Omron CX-Programmer project 新專案 (CX-Programmer 9.54)

# PLC 新PLC1: CJ2M CPU31
I/O table (CPU CJ2M-CPU31): rack 0 slot 0 CJ1W-SCU41-V1; rack 0 slot 1 CJ1W-ID231; rack 0 slot 2 CJ1W-ID231; rack 0 slot 3 CJ1W-OD231; rack 0 slot 4 CJ1W-ID211; rack 0 slot 11 CJ2M-EIP21

## Global symbols (name address type ; comment)
3.10 BOOL  ; SG舵機上感測器
3.11 BOOL  ; SG舵機下感測器
3.12 BOOL  ; PH舵機上感測器
3.13 BOOL  ; PH舵機下感測器
3.14 BOOL  ; UV舵機上感測器
3.15 BOOL  ; UV舵機下感測器
4.00 BOOL  ; SG隔膜清洗
4.01 BOOL  ; PH隔膜清洗
4.02 BOOL  ; UV隔膜清洗
4.03 BOOL  ; UV補純水
4.04 BOOL  ; SG抽液馬達
4.08 BOOL  ; 純水馬達
4.09 BOOL  ; SG舵機
4.10 BOOL  ; PH舵機
4.11 BOOL  ; UV舵機
4.12 BOOL  ; UV攪拌器
50.00 BOOL  ; 重置
50.01 BOOL  ; UV整數加
50.02 BOOL  ; UV分數加
50.03 BOOL  ; 六千
50.04 BOOL  ; 指定
50.05 BOOL  ; 回推
50.06 BOOL  ; 零點
50.07 BOOL  ; 方向
50.08 BOOL  ; 左轉
50.09 BOOL  ; 中間
50.10 BOOL  ; 右轉
50.11 BOOL  ; 速度
5.00 BOOL  ; 綠燈
5.01 BOOL  ; 橘燈
5.02 BOOL  ; 紅燈
5.03 BOOL  ; 蜂鳴器
6.00 BOOL  ; 純水低液位
6.01 BOOL  ; 純水高液位
D0 CHANNEL  ; Robot起點
D1 CHANNEL  ; Robot終點
D100 CHANNEL  ; SG平台狀態
D2 CHANNEL  ; Robot目前位置
D200 CHANNEL  ; PH平台狀態
D20001 CHANNEL  ; Seat1
D20002 CHANNEL  ; Seat2
D20003 CHANNEL  ; Seat3
D3 CHANNEL  ; 開蓋旗標
D300 CHANNEL  ; UV平台狀態
D301 CHANNEL  ; 針閥排隊
D310 CHANNEL  ; 針一狀態
D311 CHANNEL  ; 針一是否校正液
D312 CHANNEL  ; 針一整數次數
D313 CHANNEL  ; 針一分數高位
D314 CHANNEL  ; 針一分數低位
D315 CHANNEL  ; 針一指令傳送成功
D320 CHANNEL  ; 針二狀態
D321 CHANNEL  ; 針二是否校正液
D322 CHANNEL  ; 針二整數次數
D323 CHANNEL  ; 針二分數高位
D324 CHANNEL  ; 針二分數低位
D325 CHANNEL  ; 針二指令傳送成功
D330 CHANNEL  ; 針三狀態
D331 CHANNEL  ; 針三是否校正液
D332 CHANNEL  ; 針三整數次數
D333 CHANNEL  ; 針三分數高位
D334 CHANNEL  ; 針三分數低位
D335 CHANNEL  ; 針三指令傳送成功
D9998 CHANNEL  ; 稼動綠燈號
D9999 CHANNEL  ; 稼動率蜂鳴器
H100.00 BOOL  ; SG空閒
H100.01 BOOL  ; SG杯子送入
H100.02 BOOL  ; SG下舵機
H100.03 BOOL  ; SG抽樣品
H100.04 BOOL  ; SG等待
H100.05 BOOL  ; SG讀值中
H100.06 BOOL  ; SG起舵機
H100.07 BOOL  ; SG等移出
H100.08 BOOL  ; SG已移出
H100.09 BOOL  ; SG清洗
H100.10 BOOL  ; 清洗完畢
H150.01 BOOL  ; SG瓶子放入
H150.02 BOOL  ; SG下舵機
H150.03 BOOL  ; SG抽酸洗液
H150.04 BOOL  ; SG起舵機
H150.05 BOOL  ; SG等移出
H150.06 BOOL  ; SG已移出
H150.07 BOOL  ; SG清洗
H150.08 BOOL  ; SG清洗完畢
H200.00 BOOL  ; PH空閒
H200.01 BOOL  ; PH杯子送入
H200.02 BOOL  ; PH下舵機
H200.03 BOOL  ; PH等待
H200.04 BOOL  ; PH讀值中
H200.05 BOOL  ; PH起舵機
H200.06 BOOL  ; PH等移出
H200.07 BOOL  ; PH已移出
H200.08 BOOL  ; PH清洗
H200.09 BOOL  ; PH清洗完畢
H250.01 BOOL  ; PH水洗
H250.02 BOOL  ; PH水洗完畢
H300.00 BOOL  ; UV空閒
H300.01 BOOL  ; UV杯子送入
H300.02 BOOL  ; UV下舵機
H300.03 BOOL  ; UV樣品初始化
H300.04 BOOL  ; UV排液
H300.05 BOOL  ; UV注水
H300.06 BOOL  ; UV排乾
H300.07 BOOL  ; UV打歸零緩衝液
H300.08 BOOL  ; UV排液
H300.09 BOOL  ; UV等待
H300.10 BOOL  ; UV設定波長歸零
H300.11 BOOL  ; UV注水
H300.12 BOOL  ; UV排液
H300.13 BOOL  ; UV整數取樣
H300.14 BOOL  ; UV分數取樣
H300.15 BOOL  ; UV抽液
H301.00 BOOL  ; UV等待
H301.01 BOOL  ; UV讀值
H301.02 BOOL  ; UV起舵機
H301.03 BOOL  ; UV等待移出
H301.04 BOOL  ; UV已移出
H301.05 BOOL  ; UV針閥清洗
H301.06 BOOL  ; UV排乾
H301.07 BOOL  ; UV補水
H301.08 BOOL  ; UV排乾
H301.09 BOOL  ; UV清洗完畢
W0.00 BOOL  ; 針閥1初始化
W0.01 BOOL  ; 針閥二初始化
W300.00 BOOL  ; 樣品初始化開始
W300.01 BOOL  ; 樣品初始化中
W300.02 BOOL  ; 樣品初始化完成
W300.03 BOOL  ; 分數取樣完成
W301.00 BOOL  ; 打緩衝液開始
W301.01 BOOL  ; 打緩衝液中
W301.02 BOOL  ; 打緩衝液完成
W302.00 BOOL  ; UV整數取樣開始
W302.01 BOOL  ; UV整數取樣中
W302.02 BOOL  ; UV整數取樣完成
W303.00 BOOL  ; UV分數取樣開始
W303.01 BOOL  ; UV分數取樣中
W303.02 BOOL  ; UV分數取樣完成
W304.00 BOOL  ; 針閥清洗
W304.01 BOOL  ; 針閥清洗中
W304.02 BOOL  ; 針閥清洗完成
W304.03 BOOL  ; 補水
W305.00 BOOL  ; 二次補水
W305.01 BOOL  ; 三次補水
W306.00 BOOL  ; 清洗二次補水
W306.01 BOOL  ; 清洗三次補水

## Program 新增程式1 (cyclic task 0)
Local symbols
FFFF CHANNEL
md BOOL

### Section Platform1_SG

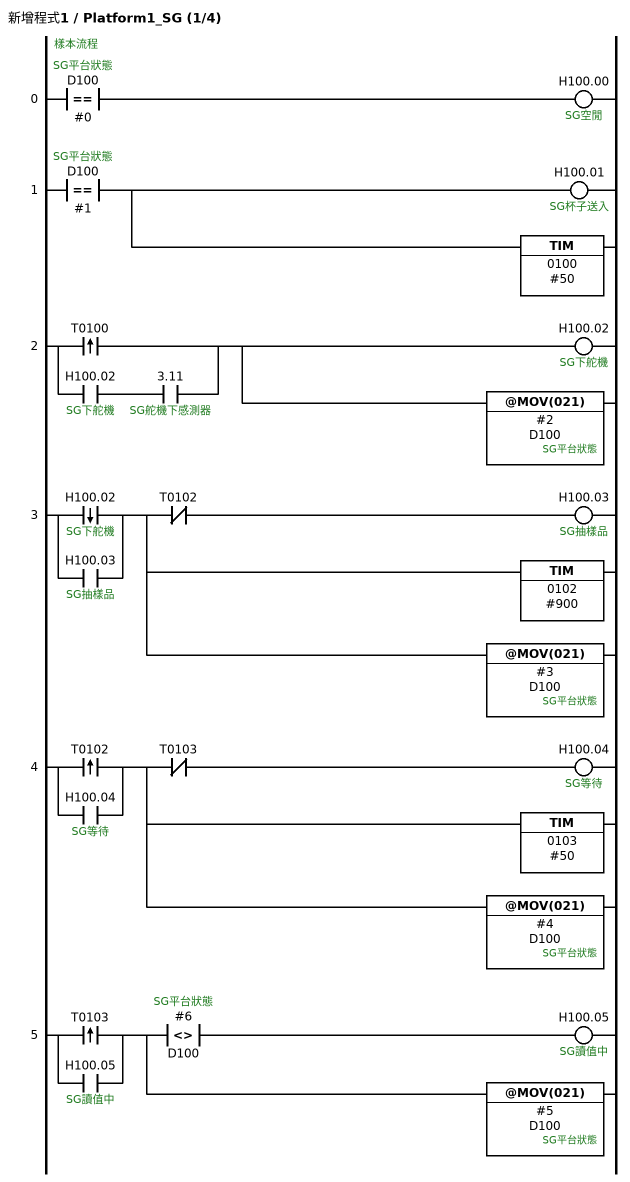
; rung 0: 樣本流程
LD=(300) D100 #0  ; SG平台狀態
OUT H100.00  ; SG空閒
; rung 1
LD=(300) D100 #1  ; SG平台狀態
OUT H100.01  ; SG杯子送入
TIM 0100 #50
; rung 2
@LD T0100
LD H100.02  ; SG下舵機
AND 3.11  ; SG舵機下感測器
ORLD
OUT H100.02  ; SG下舵機
@MOV(021) #2 D100  ; SG平台狀態
; rung 3
%LD H100.02  ; SG下舵機
OR H100.03  ; SG抽樣品
OUT TR0
ANDNOT T0102
OUT H100.03  ; SG抽樣品
LD TR0
TIM 0102 #900
@MOV(021) #3 D100  ; SG平台狀態
; rung 4
@LD T0102
OR H100.04  ; SG等待
OUT TR0
ANDNOT T0103
OUT H100.04  ; SG等待
LD TR0
TIM 0103 #50
@MOV(021) #4 D100  ; SG平台狀態
; rung 5
@LD T0103
OR H100.05  ; SG讀值中
OUT TR0
AND<>(305) #6 D100  ; SG平台狀態
OUT H100.05  ; SG讀值中
LD TR0
@MOV(021) #5 D100  ; SG平台狀態

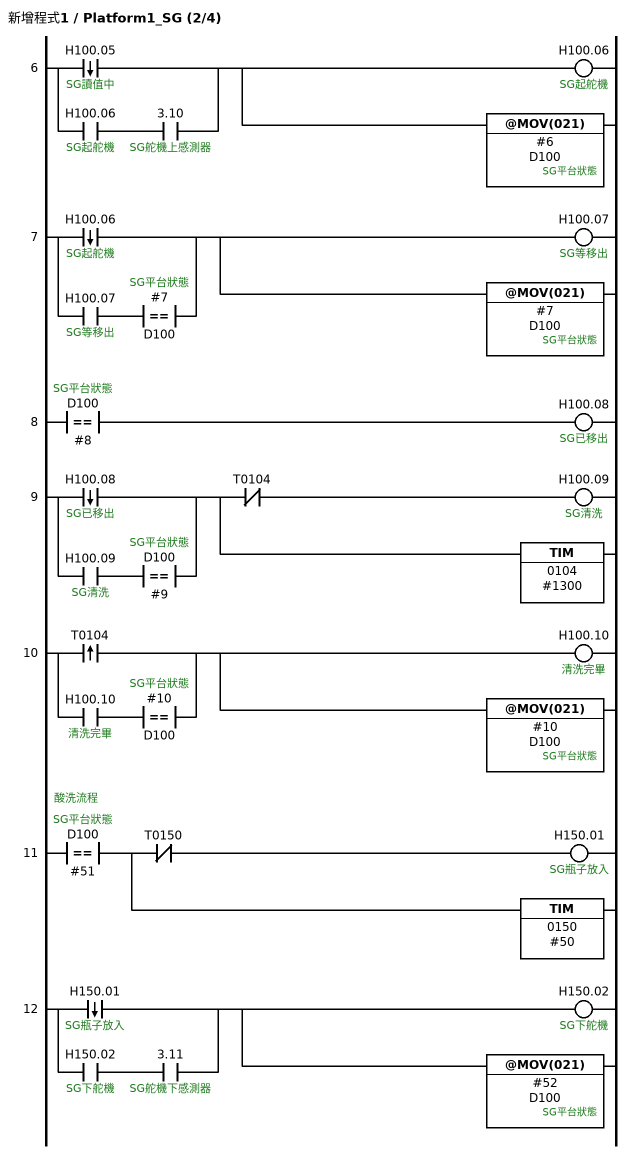
; rung 6
%LD H100.05  ; SG讀值中
LD H100.06  ; SG起舵機
AND 3.10  ; SG舵機上感測器
ORLD
OUT H100.06  ; SG起舵機
@MOV(021) #6 D100  ; SG平台狀態
; rung 7
%LD H100.06  ; SG起舵機
LD H100.07  ; SG等移出
AND=(300) #7 D100  ; SG平台狀態
ORLD
OUT H100.07  ; SG等移出
@MOV(021) #7 D100  ; SG平台狀態
; rung 8
LD=(300) D100 #8  ; SG平台狀態
OUT H100.08  ; SG已移出
; rung 9
%LD H100.08  ; SG已移出
LD H100.09  ; SG清洗
AND=(300) D100 #9  ; SG平台狀態
ORLD
OUT TR0
ANDNOT T0104
OUT H100.09  ; SG清洗
LD TR0
TIM 0104 #1300
; rung 10
@LD T0104
LD H100.10  ; 清洗完畢
AND=(300) #10 D100  ; SG平台狀態
ORLD
OUT H100.10  ; 清洗完畢
@MOV(021) #10 D100  ; SG平台狀態
; rung 11: 酸洗流程
LD=(300) D100 #51  ; SG平台狀態
OUT TR0
ANDNOT T0150
OUT H150.01  ; SG瓶子放入
LD TR0
TIM 0150 #50
; rung 12
%LD H150.01  ; SG瓶子放入
LD H150.02  ; SG下舵機
AND 3.11  ; SG舵機下感測器
ORLD
OUT H150.02  ; SG下舵機
@MOV(021) #52 D100  ; SG平台狀態

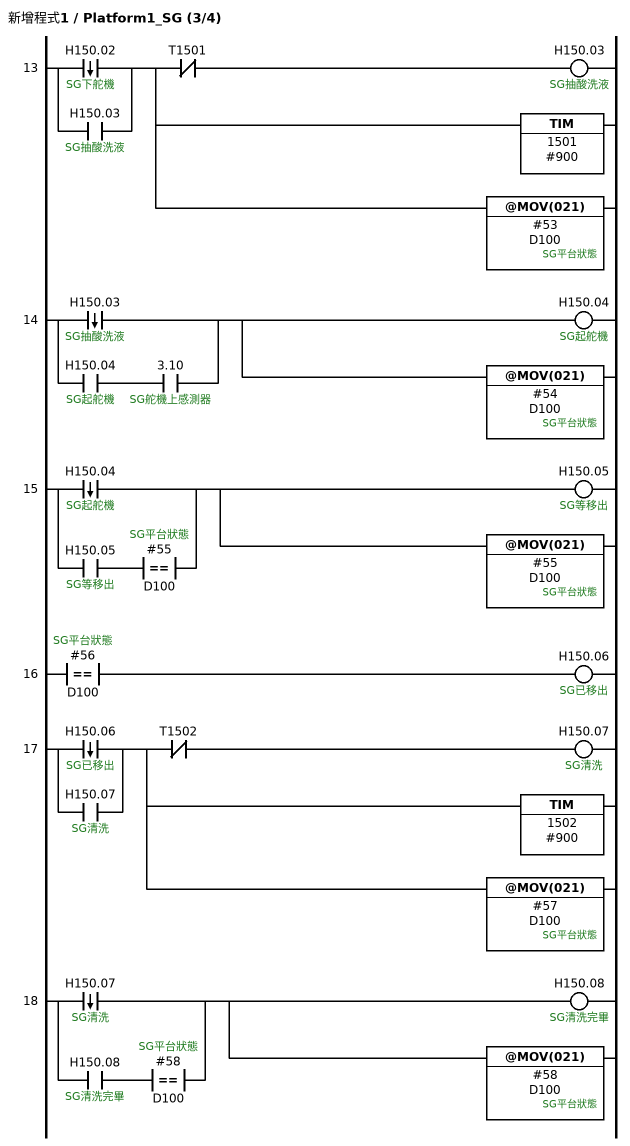
; rung 13
%LD H150.02  ; SG下舵機
OR H150.03  ; SG抽酸洗液
OUT TR0
ANDNOT T1501
OUT H150.03  ; SG抽酸洗液
LD TR0
TIM 1501 #900
@MOV(021) #53 D100  ; SG平台狀態
; rung 14
%LD H150.03  ; SG抽酸洗液
LD H150.04  ; SG起舵機
AND 3.10  ; SG舵機上感測器
ORLD
OUT H150.04  ; SG起舵機
@MOV(021) #54 D100  ; SG平台狀態
; rung 15
%LD H150.04  ; SG起舵機
LD H150.05  ; SG等移出
AND=(300) #55 D100  ; SG平台狀態
ORLD
OUT H150.05  ; SG等移出
@MOV(021) #55 D100  ; SG平台狀態
; rung 16
LD=(300) #56 D100  ; SG平台狀態
OUT H150.06  ; SG已移出
; rung 17
%LD H150.06  ; SG已移出
OR H150.07  ; SG清洗
OUT TR0
ANDNOT T1502
OUT H150.07  ; SG清洗
LD TR0
TIM 1502 #900
@MOV(021) #57 D100  ; SG平台狀態
; rung 18
%LD H150.07  ; SG清洗
LD H150.08  ; SG清洗完畢
AND=(300) #58 D100  ; SG平台狀態
ORLD
OUT H150.08  ; SG清洗完畢
@MOV(021) #58 D100  ; SG平台狀態

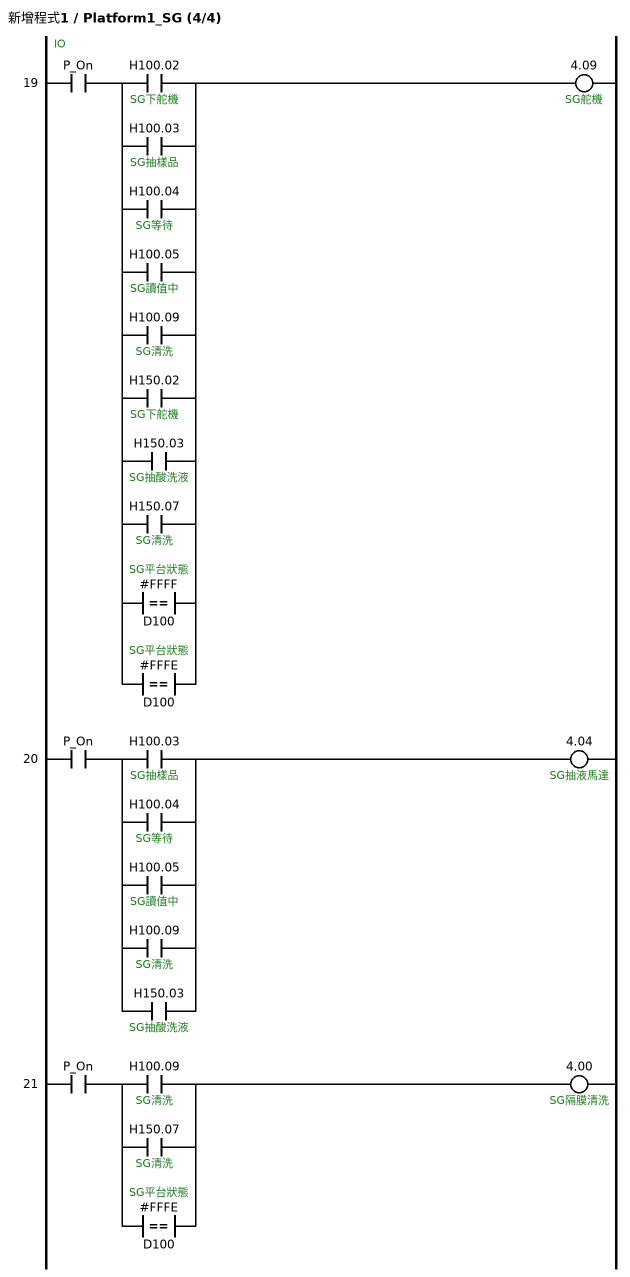
; rung 19: IO
LD P_On
LD H100.02  ; SG下舵機
OR H100.03  ; SG抽樣品
OR H100.04  ; SG等待
OR H100.05  ; SG讀值中
OR H100.09  ; SG清洗
OR H150.02  ; SG下舵機
OR H150.03  ; SG抽酸洗液
OR H150.07  ; SG清洗
OR=(300) #FFFF D100  ; SG平台狀態
OR=(300) #FFFE D100  ; SG平台狀態
ANDLD
OUT 4.09  ; SG舵機
; rung 20
LD P_On
LD H100.03  ; SG抽樣品
OR H100.04  ; SG等待
OR H100.05  ; SG讀值中
OR H100.09  ; SG清洗
OR H150.03  ; SG抽酸洗液
ANDLD
OUT 4.04  ; SG抽液馬達
; rung 21
LD P_On
LD H100.09  ; SG清洗
OR H150.07  ; SG清洗
OR=(300) #FFFE D100  ; SG平台狀態
ANDLD
OUT 4.00  ; SG隔膜清洗

### Section Platform2_PH

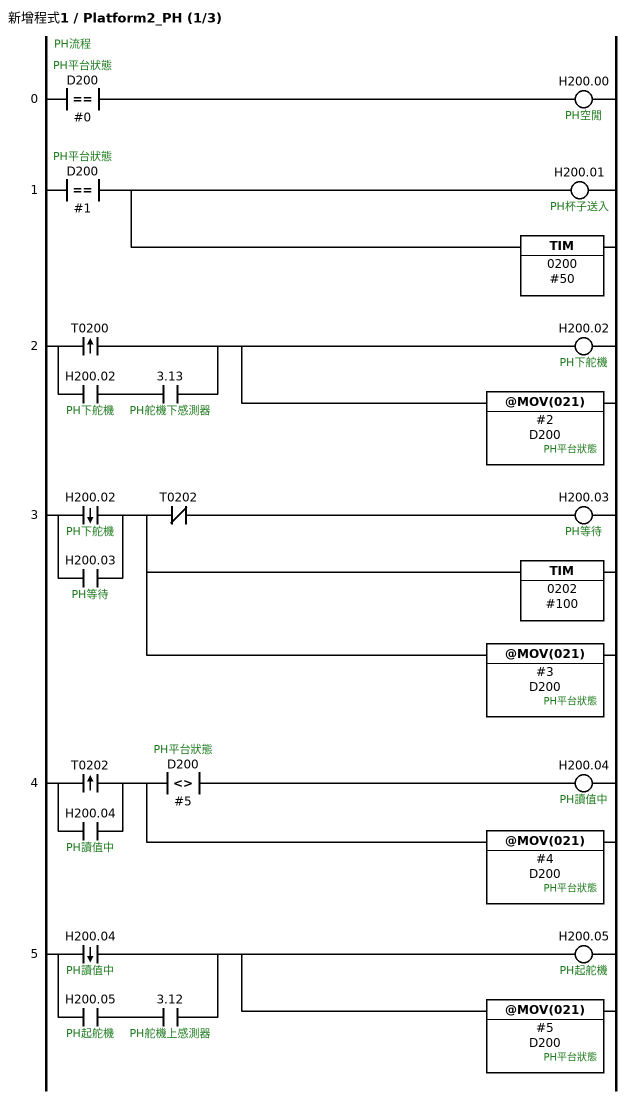
; rung 0: PH流程
LD=(300) D200 #0  ; PH平台狀態
OUT H200.00  ; PH空閒
; rung 1
LD=(300) D200 #1  ; PH平台狀態
OUT H200.01  ; PH杯子送入
TIM 0200 #50
; rung 2
@LD T0200
LD H200.02  ; PH下舵機
AND 3.13  ; PH舵機下感測器
ORLD
OUT H200.02  ; PH下舵機
@MOV(021) #2 D200  ; PH平台狀態
; rung 3
%LD H200.02  ; PH下舵機
OR H200.03  ; PH等待
OUT TR0
ANDNOT T0202
OUT H200.03  ; PH等待
LD TR0
TIM 0202 #100
@MOV(021) #3 D200  ; PH平台狀態
; rung 4
@LD T0202
OR H200.04  ; PH讀值中
OUT TR0
AND<>(305) D200 #5  ; PH平台狀態
OUT H200.04  ; PH讀值中
LD TR0
@MOV(021) #4 D200  ; PH平台狀態
; rung 5
%LD H200.04  ; PH讀值中
LD H200.05  ; PH起舵機
AND 3.12  ; PH舵機上感測器
ORLD
OUT H200.05  ; PH起舵機
@MOV(021) #5 D200  ; PH平台狀態

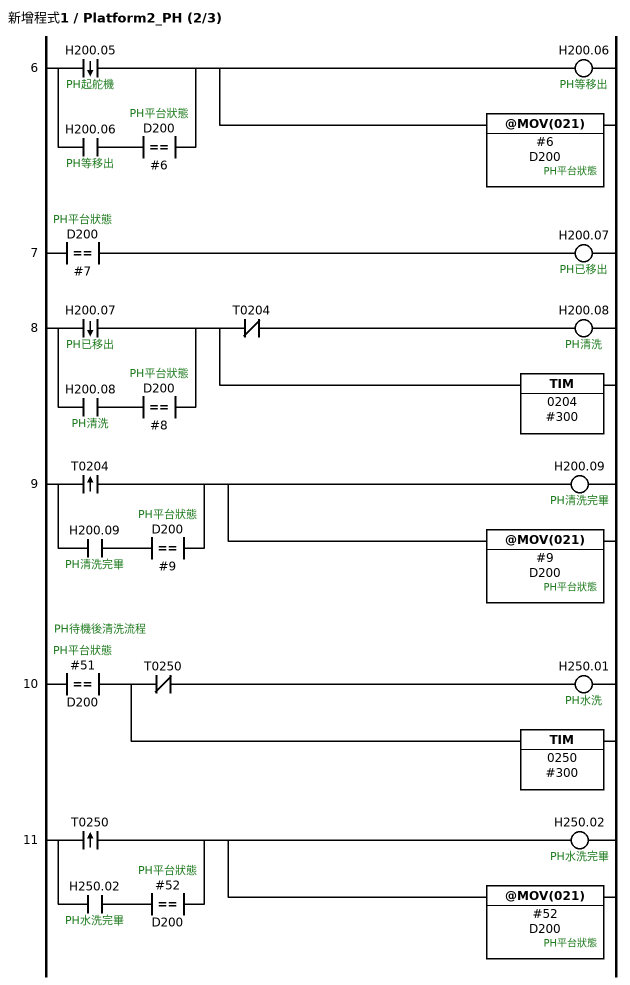
; rung 6
%LD H200.05  ; PH起舵機
LD H200.06  ; PH等移出
AND=(300) D200 #6  ; PH平台狀態
ORLD
OUT H200.06  ; PH等移出
@MOV(021) #6 D200  ; PH平台狀態
; rung 7
LD=(300) D200 #7  ; PH平台狀態
OUT H200.07  ; PH已移出
; rung 8
%LD H200.07  ; PH已移出
LD H200.08  ; PH清洗
AND=(300) D200 #8  ; PH平台狀態
ORLD
OUT TR0
ANDNOT T0204
OUT H200.08  ; PH清洗
LD TR0
TIM 0204 #300
; rung 9
@LD T0204
LD H200.09  ; PH清洗完畢
AND=(300) D200 #9  ; PH平台狀態
ORLD
OUT H200.09  ; PH清洗完畢
@MOV(021) #9 D200  ; PH平台狀態
; rung 10: PH待機後清洗流程
LD=(300) #51 D200  ; PH平台狀態
OUT TR0
ANDNOT T0250
OUT H250.01  ; PH水洗
LD TR0
TIM 0250 #300
; rung 11
@LD T0250
LD H250.02  ; PH水洗完畢
AND=(300) #52 D200  ; PH平台狀態
ORLD
OUT H250.02  ; PH水洗完畢
@MOV(021) #52 D200  ; PH平台狀態

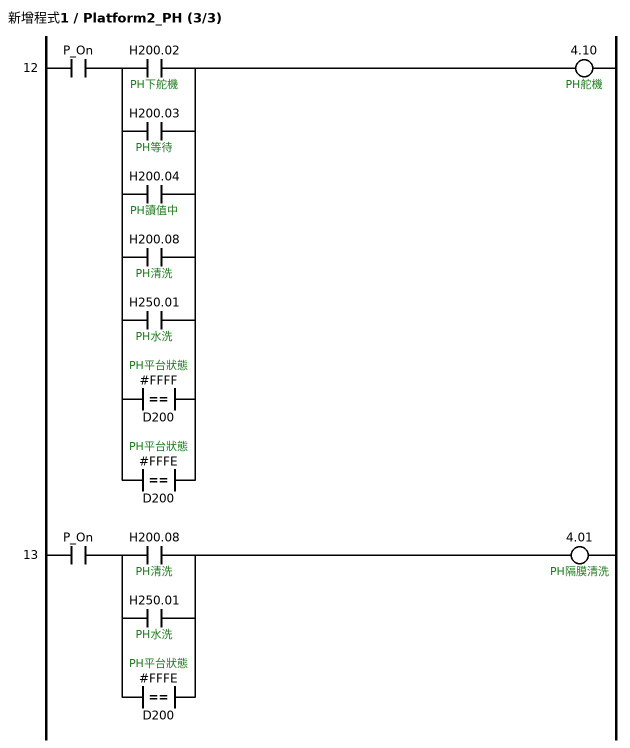
; rung 12
LD P_On
LD H200.02  ; PH下舵機
OR H200.03  ; PH等待
OR H200.04  ; PH讀值中
OR H200.08  ; PH清洗
OR H250.01  ; PH水洗
OR=(300) #FFFF D200  ; PH平台狀態
OR=(300) #FFFE D200  ; PH平台狀態
ANDLD
OUT 4.10  ; PH舵機
; rung 13
LD P_On
LD H200.08  ; PH清洗
OR H250.01  ; PH水洗
OR=(300) #FFFE D200  ; PH平台狀態
ANDLD
OUT 4.01  ; PH隔膜清洗

### Section Platform3_UV

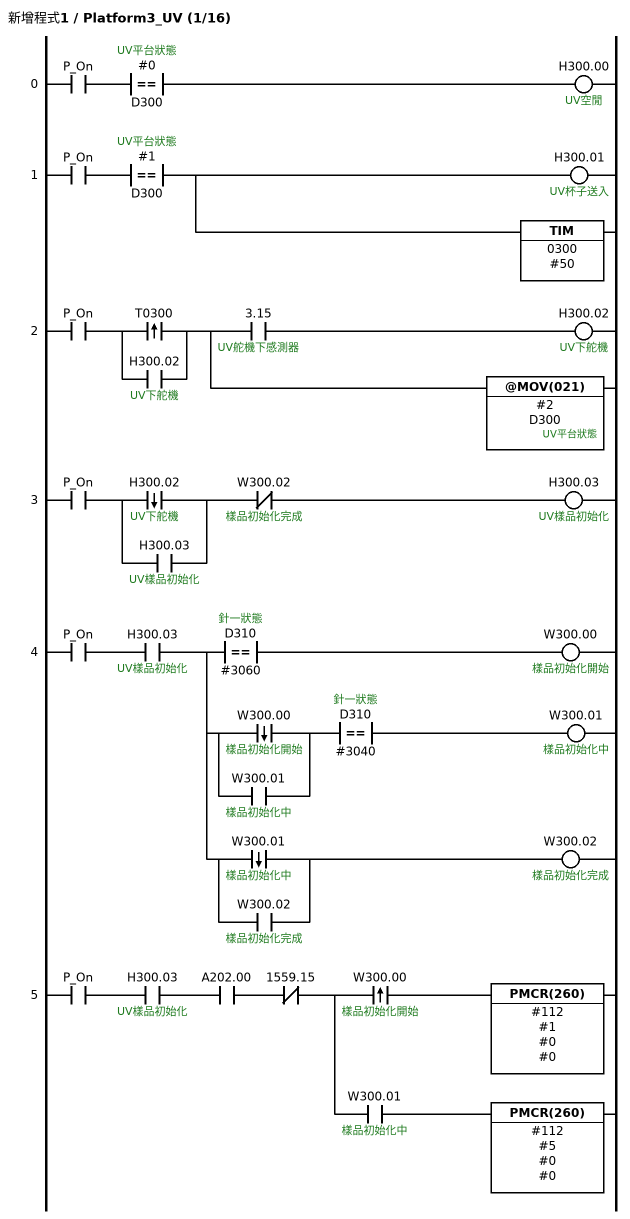
; rung 0
LD P_On
AND=(300) #0 D300  ; UV平台狀態
OUT H300.00  ; UV空閒
; rung 1
LD P_On
AND=(300) #1 D300  ; UV平台狀態
OUT H300.01  ; UV杯子送入
TIM 0300 #50
; rung 2
LD P_On
@LD T0300
OR H300.02  ; UV下舵機
ANDLD
OUT TR0
AND 3.15  ; UV舵機下感測器
OUT H300.02  ; UV下舵機
LD TR0
@MOV(021) #2 D300  ; UV平台狀態
; rung 3
LD P_On
%LD H300.02  ; UV下舵機
OR H300.03  ; UV樣品初始化
ANDLD
ANDNOT W300.02  ; 樣品初始化完成
OUT H300.03  ; UV樣品初始化
; rung 4
LD P_On
AND H300.03  ; UV樣品初始化
OUT TR0
AND=(300) D310 #3060  ; 針一狀態
OUT W300.00  ; 樣品初始化開始
LD TR0
%LD W300.00  ; 樣品初始化開始
OR W300.01  ; 樣品初始化中
ANDLD
AND=(300) D310 #3040  ; 針一狀態
OUT W300.01  ; 樣品初始化中
LD TR0
%LD W300.01  ; 樣品初始化中
OR W300.02  ; 樣品初始化完成
ANDLD
OUT W300.02  ; 樣品初始化完成
; rung 5
LD P_On
AND H300.03  ; UV樣品初始化
AND A202.00
ANDNOT 1559.15
OUT TR0
@AND W300.00  ; 樣品初始化開始
PMCR(260) #112 #1 #0 #0
LD TR0
AND W300.01  ; 樣品初始化中
PMCR(260) #112 #5 #0 #0

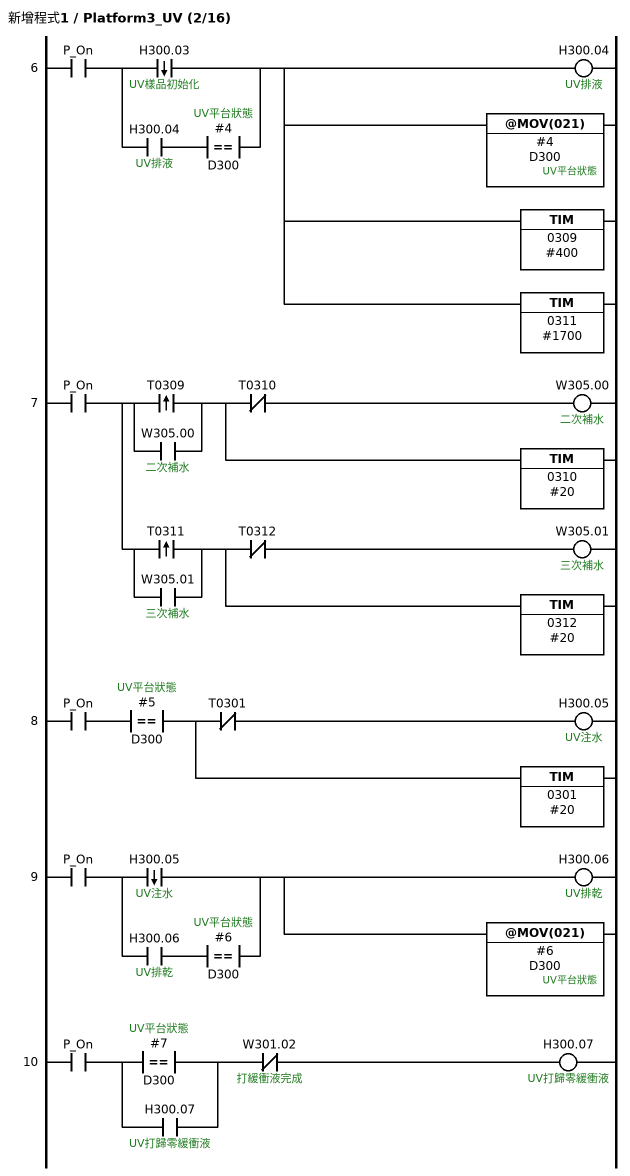
; rung 6
LD P_On
%LD H300.03  ; UV樣品初始化
LD H300.04  ; UV排液
AND=(300) #4 D300  ; UV平台狀態
ORLD
ANDLD
OUT H300.04  ; UV排液
@MOV(021) #4 D300  ; UV平台狀態
TIM 0309 #400
TIM 0311 #1700
; rung 7
LD P_On
OUT TR0
@LD T0309
OR W305.00  ; 二次補水
ANDLD
OUT TR1
ANDNOT T0310
OUT W305.00  ; 二次補水
LD TR1
TIM 0310 #20
LD TR0
@LD T0311
OR W305.01  ; 三次補水
ANDLD
OUT TR0
ANDNOT T0312
OUT W305.01  ; 三次補水
LD TR0
TIM 0312 #20
; rung 8
LD P_On
AND=(300) #5 D300  ; UV平台狀態
OUT TR0
ANDNOT T0301
OUT H300.05  ; UV注水
LD TR0
TIM 0301 #20
; rung 9
LD P_On
%LD H300.05  ; UV注水
LD H300.06  ; UV排乾
AND=(300) #6 D300  ; UV平台狀態
ORLD
ANDLD
OUT H300.06  ; UV排乾
@MOV(021) #6 D300  ; UV平台狀態
; rung 10
LD P_On
LD=(300) #7 D300  ; UV平台狀態
OR H300.07  ; UV打歸零緩衝液
ANDLD
ANDNOT W301.02  ; 打緩衝液完成
OUT H300.07  ; UV打歸零緩衝液

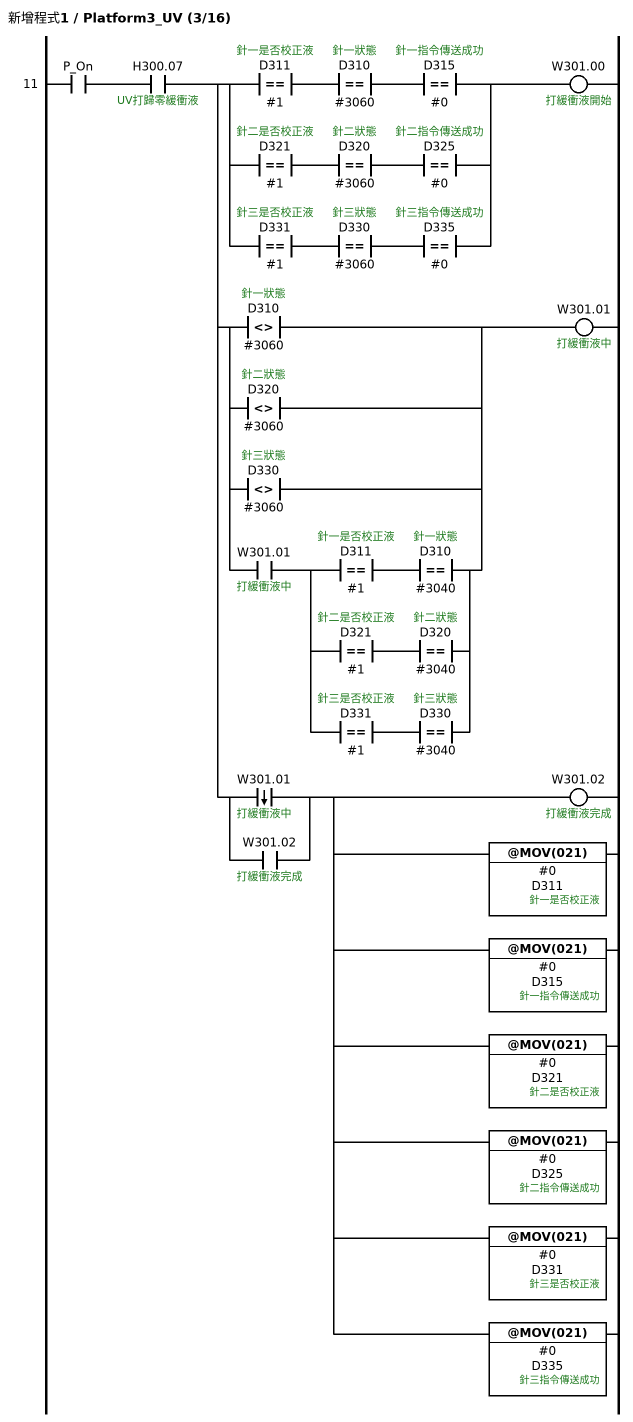
; rung 11
LD P_On
AND H300.07  ; UV打歸零緩衝液
OUT TR0
LD=(300) D311 #1  ; 針一是否校正液
AND=(300) D310 #3060  ; 針一狀態
AND=(300) D315 #0  ; 針一指令傳送成功
LD=(300) D321 #1  ; 針二是否校正液
AND=(300) D320 #3060  ; 針二狀態
AND=(300) D325 #0  ; 針二指令傳送成功
ORLD
LD=(300) D331 #1  ; 針三是否校正液
AND=(300) D330 #3060  ; 針三狀態
AND=(300) D335 #0  ; 針三指令傳送成功
ORLD
ANDLD
OUT W301.00  ; 打緩衝液開始
LD TR0
LD<>(305) D310 #3060  ; 針一狀態
OR<>(305) D320 #3060  ; 針二狀態
OR<>(305) D330 #3060  ; 針三狀態
LD W301.01  ; 打緩衝液中
LD=(300) D311 #1  ; 針一是否校正液
AND=(300) D310 #3040  ; 針一狀態
LD=(300) D321 #1  ; 針二是否校正液
AND=(300) D320 #3040  ; 針二狀態
ORLD
LD=(300) D331 #1  ; 針三是否校正液
AND=(300) D330 #3040  ; 針三狀態
ORLD
ANDLD
ORLD
ANDLD
OUT W301.01  ; 打緩衝液中
LD TR0
%LD W301.01  ; 打緩衝液中
OR W301.02  ; 打緩衝液完成
ANDLD
OUT W301.02  ; 打緩衝液完成
@MOV(021) #0 D311  ; 針一是否校正液
@MOV(021) #0 D315  ; 針一指令傳送成功
@MOV(021) #0 D321  ; 針二是否校正液
@MOV(021) #0 D325  ; 針二指令傳送成功
@MOV(021) #0 D331  ; 針三是否校正液
@MOV(021) #0 D335  ; 針三指令傳送成功

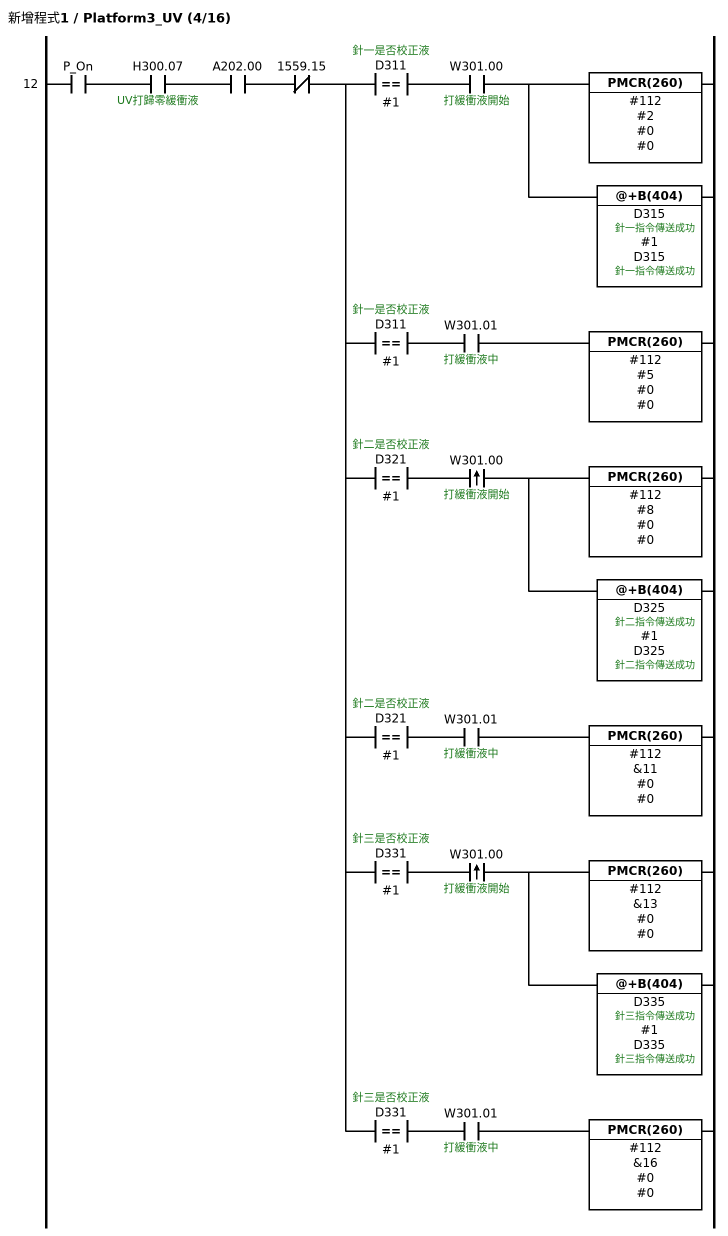
; rung 12
LD P_On
AND H300.07  ; UV打歸零緩衝液
AND A202.00
ANDNOT 1559.15
OUT TR0
AND=(300) D311 #1  ; 針一是否校正液
AND W301.00  ; 打緩衝液開始
PMCR(260) #112 #2 #0 #0
@+B(404) D315 #1 D315  ; 針一指令傳送成功
LD TR0
AND=(300) D311 #1  ; 針一是否校正液
AND W301.01  ; 打緩衝液中
PMCR(260) #112 #5 #0 #0
LD TR0
AND=(300) D321 #1  ; 針二是否校正液
@AND W301.00  ; 打緩衝液開始
PMCR(260) #112 #8 #0 #0
@+B(404) D325 #1 D325  ; 針二指令傳送成功
LD TR0
AND=(300) D321 #1  ; 針二是否校正液
AND W301.01  ; 打緩衝液中
PMCR(260) #112 &11 #0 #0
LD TR0
AND=(300) D331 #1  ; 針三是否校正液
@AND W301.00  ; 打緩衝液開始
PMCR(260) #112 &13 #0 #0
@+B(404) D335 #1 D335  ; 針三指令傳送成功
LD TR0
AND=(300) D331 #1  ; 針三是否校正液
AND W301.01  ; 打緩衝液中
PMCR(260) #112 &16 #0 #0

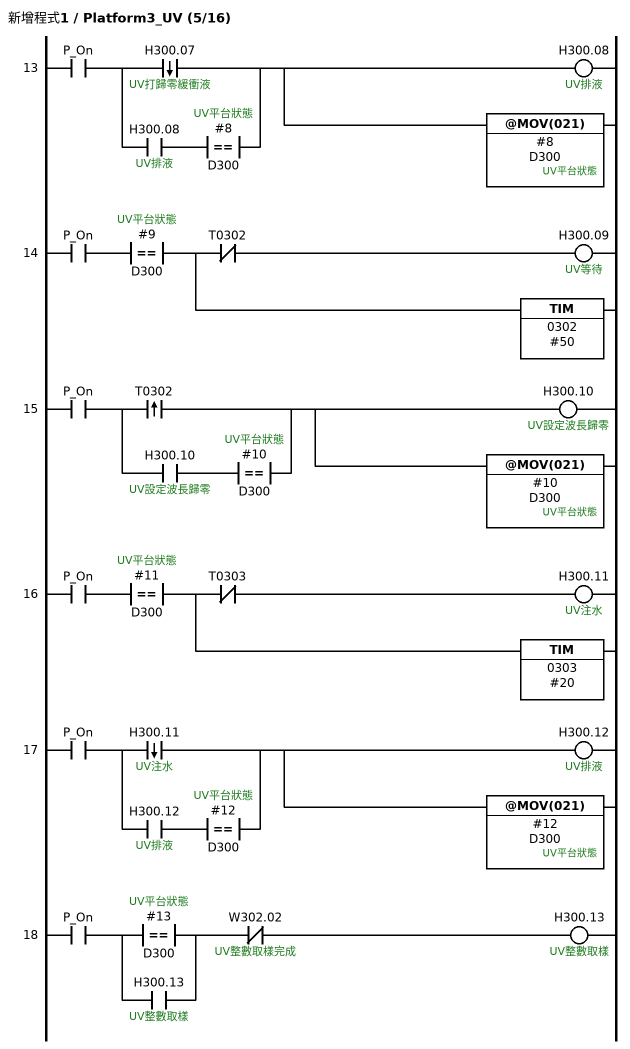
; rung 13
LD P_On
%LD H300.07  ; UV打歸零緩衝液
LD H300.08  ; UV排液
AND=(300) #8 D300  ; UV平台狀態
ORLD
ANDLD
OUT H300.08  ; UV排液
@MOV(021) #8 D300  ; UV平台狀態
; rung 14
LD P_On
AND=(300) #9 D300  ; UV平台狀態
OUT TR0
ANDNOT T0302
OUT H300.09  ; UV等待
LD TR0
TIM 0302 #50
; rung 15
LD P_On
@LD T0302
LD H300.10  ; UV設定波長歸零
AND=(300) #10 D300  ; UV平台狀態
ORLD
ANDLD
OUT H300.10  ; UV設定波長歸零
@MOV(021) #10 D300  ; UV平台狀態
; rung 16
LD P_On
AND=(300) #11 D300  ; UV平台狀態
OUT TR0
ANDNOT T0303
OUT H300.11  ; UV注水
LD TR0
TIM 0303 #20
; rung 17
LD P_On
%LD H300.11  ; UV注水
LD H300.12  ; UV排液
AND=(300) #12 D300  ; UV平台狀態
ORLD
ANDLD
OUT H300.12  ; UV排液
@MOV(021) #12 D300  ; UV平台狀態
; rung 18
LD P_On
LD=(300) #13 D300  ; UV平台狀態
OR H300.13  ; UV整數取樣
ANDLD
ANDNOT W302.02  ; UV整數取樣完成
OUT H300.13  ; UV整數取樣

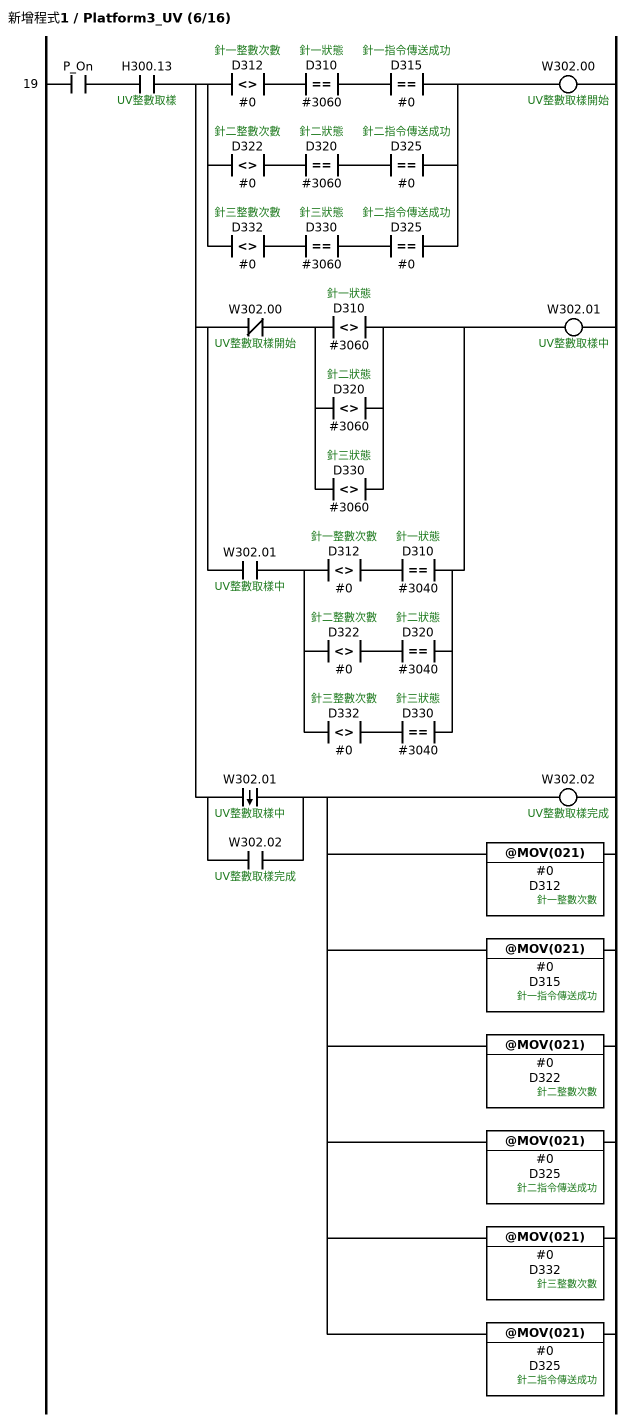
; rung 19
LD P_On
AND H300.13  ; UV整數取樣
OUT TR0
LD<>(305) D312 #0  ; 針一整數次數
AND=(300) D310 #3060  ; 針一狀態
AND=(300) D315 #0  ; 針一指令傳送成功
LD<>(305) D322 #0  ; 針二整數次數
AND=(300) D320 #3060  ; 針二狀態
AND=(300) D325 #0  ; 針二指令傳送成功
ORLD
LD<>(305) D332 #0  ; 針三整數次數
AND=(300) D330 #3060  ; 針三狀態
AND=(300) D325 #0  ; 針二指令傳送成功
ORLD
ANDLD
OUT W302.00  ; UV整數取樣開始
LD TR0
LDNOT W302.00  ; UV整數取樣開始
LD<>(305) D310 #3060  ; 針一狀態
OR<>(305) D320 #3060  ; 針二狀態
OR<>(305) D330 #3060  ; 針三狀態
ANDLD
LD W302.01  ; UV整數取樣中
LD<>(305) D312 #0  ; 針一整數次數
AND=(300) D310 #3040  ; 針一狀態
LD<>(305) D322 #0  ; 針二整數次數
AND=(300) D320 #3040  ; 針二狀態
ORLD
LD<>(305) D332 #0  ; 針三整數次數
AND=(300) D330 #3040  ; 針三狀態
ORLD
ANDLD
ORLD
ANDLD
OUT W302.01  ; UV整數取樣中
LD TR0
%LD W302.01  ; UV整數取樣中
OR W302.02  ; UV整數取樣完成
ANDLD
OUT W302.02  ; UV整數取樣完成
@MOV(021) #0 D312  ; 針一整數次數
@MOV(021) #0 D315  ; 針一指令傳送成功
@MOV(021) #0 D322  ; 針二整數次數
@MOV(021) #0 D325  ; 針二指令傳送成功
@MOV(021) #0 D332  ; 針三整數次數
@MOV(021) #0 D325  ; 針二指令傳送成功

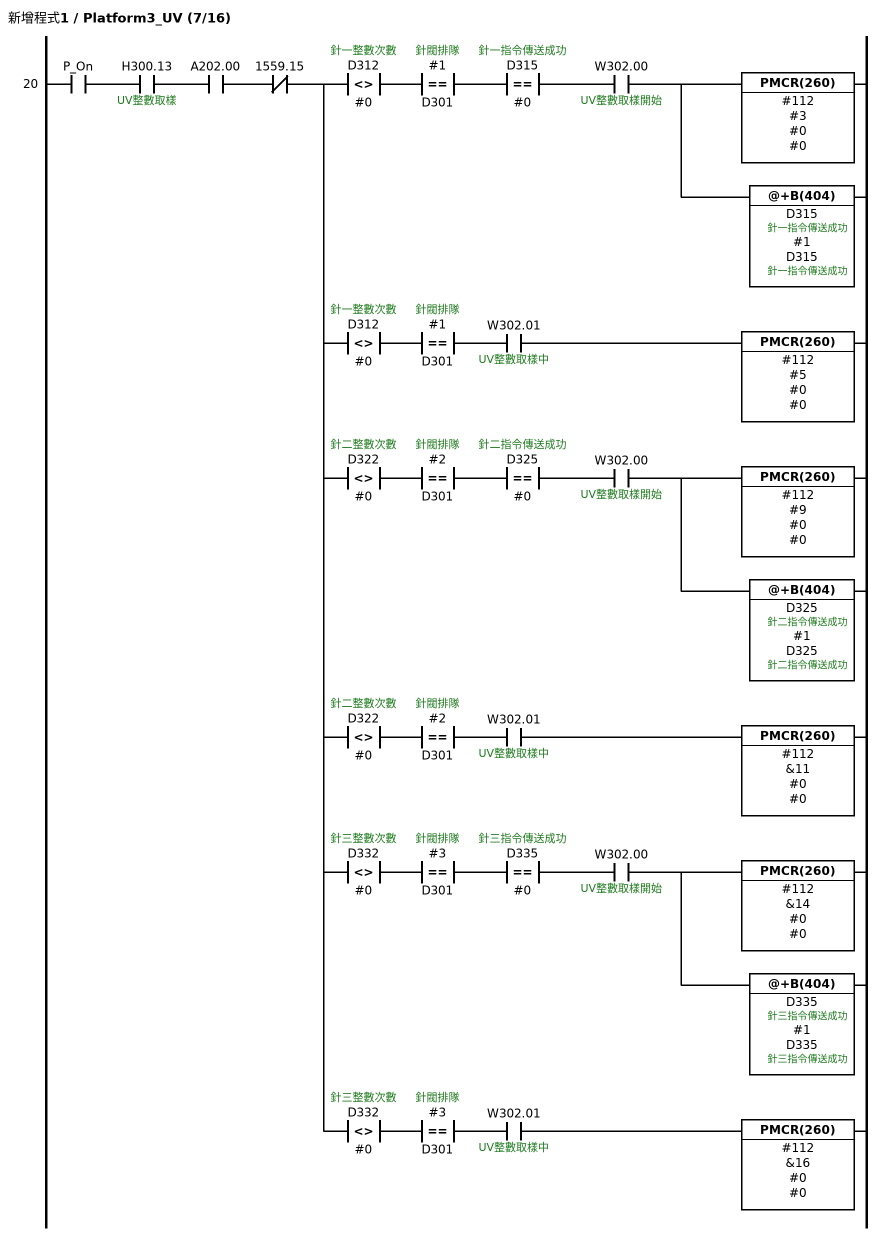
; rung 20
LD P_On
AND H300.13  ; UV整數取樣
AND A202.00
ANDNOT 1559.15
OUT TR0
AND<>(305) D312 #0  ; 針一整數次數
AND=(300) #1 D301  ; 針閥排隊
AND=(300) D315 #0  ; 針一指令傳送成功
AND W302.00  ; UV整數取樣開始
PMCR(260) #112 #3 #0 #0
@+B(404) D315 #1 D315  ; 針一指令傳送成功
LD TR0
AND<>(305) D312 #0  ; 針一整數次數
AND=(300) #1 D301  ; 針閥排隊
AND W302.01  ; UV整數取樣中
PMCR(260) #112 #5 #0 #0
LD TR0
AND<>(305) D322 #0  ; 針二整數次數
AND=(300) #2 D301  ; 針閥排隊
AND=(300) D325 #0  ; 針二指令傳送成功
AND W302.00  ; UV整數取樣開始
PMCR(260) #112 #9 #0 #0
@+B(404) D325 #1 D325  ; 針二指令傳送成功
LD TR0
AND<>(305) D322 #0  ; 針二整數次數
AND=(300) #2 D301  ; 針閥排隊
AND W302.01  ; UV整數取樣中
PMCR(260) #112 &11 #0 #0
LD TR0
AND<>(305) D332 #0  ; 針三整數次數
AND=(300) #3 D301  ; 針閥排隊
AND=(300) D335 #0  ; 針三指令傳送成功
AND W302.00  ; UV整數取樣開始
PMCR(260) #112 &14 #0 #0
@+B(404) D335 #1 D335  ; 針三指令傳送成功
LD TR0
AND<>(305) D332 #0  ; 針三整數次數
AND=(300) #3 D301  ; 針閥排隊
AND W302.01  ; UV整數取樣中
PMCR(260) #112 &16 #0 #0

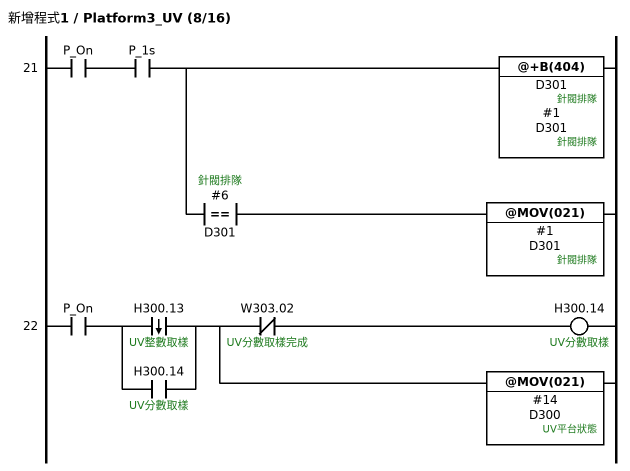
; rung 21
LD P_On
AND P_1s
@+B(404) D301 #1 D301  ; 針閥排隊
AND=(300) #6 D301  ; 針閥排隊
@MOV(021) #1 D301  ; 針閥排隊
; rung 22
LD P_On
%LD H300.13  ; UV整數取樣
OR H300.14  ; UV分數取樣
ANDLD
OUT TR0
ANDNOT W303.02  ; UV分數取樣完成
OUT H300.14  ; UV分數取樣
LD TR0
@MOV(021) #14 D300  ; UV平台狀態

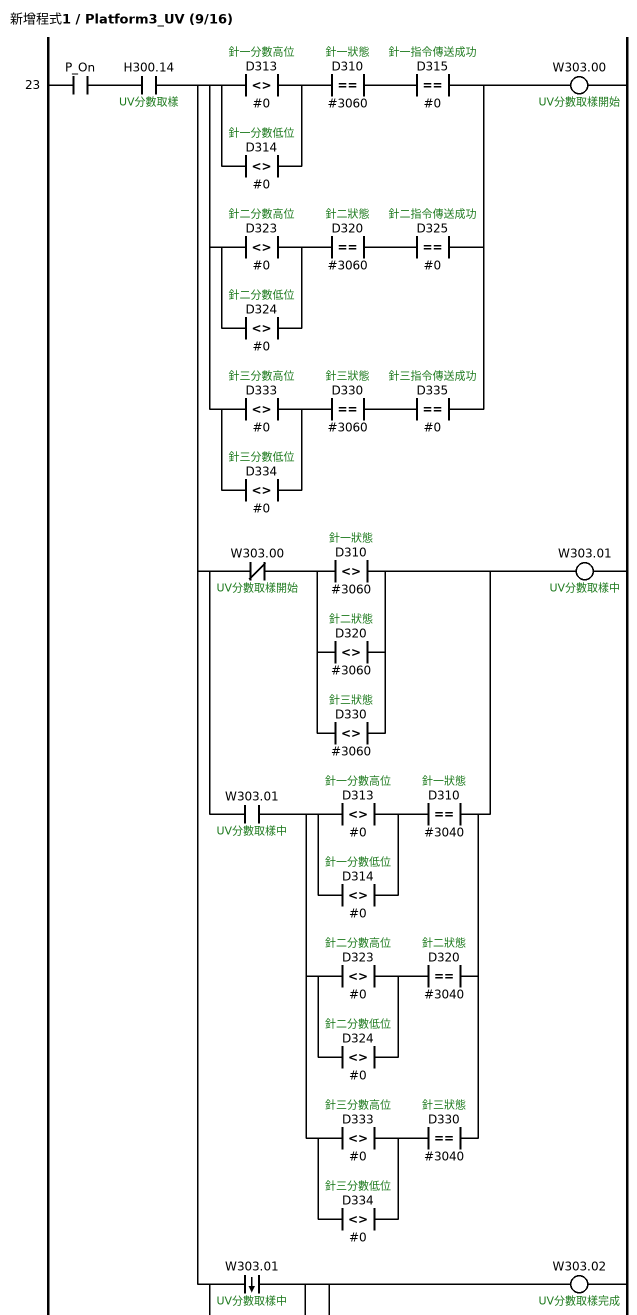

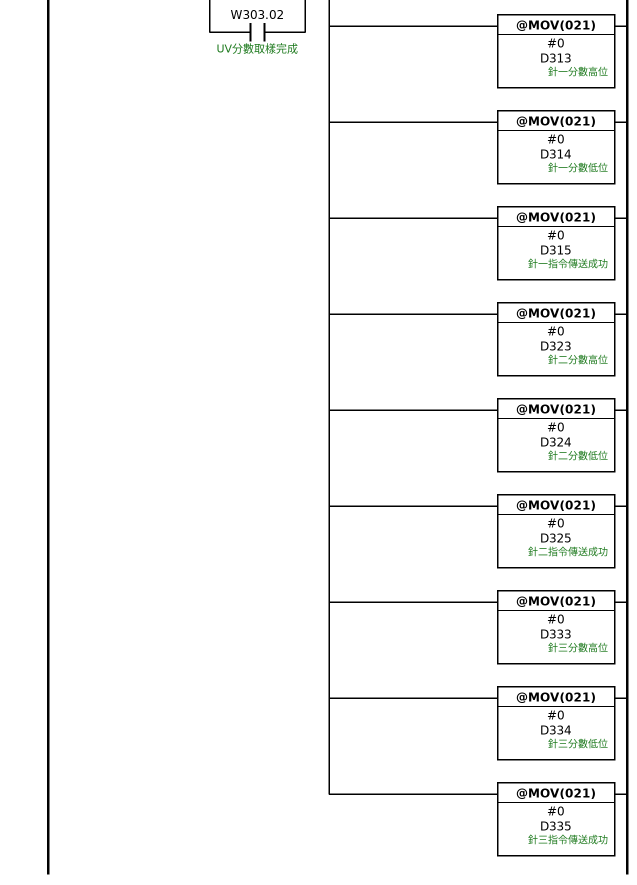
; rung 23
LD P_On
AND H300.14  ; UV分數取樣
OUT TR0
LD<>(305) D313 #0  ; 針一分數高位
OR<>(305) D314 #0  ; 針一分數低位
AND=(300) D310 #3060  ; 針一狀態
AND=(300) D315 #0  ; 針一指令傳送成功
LD<>(305) D323 #0  ; 針二分數高位
OR<>(305) D324 #0  ; 針二分數低位
AND=(300) D320 #3060  ; 針二狀態
AND=(300) D325 #0  ; 針二指令傳送成功
ORLD
LD<>(305) D333 #0  ; 針三分數高位
OR<>(305) D334 #0  ; 針三分數低位
AND=(300) D330 #3060  ; 針三狀態
AND=(300) D335 #0  ; 針三指令傳送成功
ORLD
ANDLD
OUT W303.00  ; UV分數取樣開始
LD TR0
LDNOT W303.00  ; UV分數取樣開始
LD<>(305) D310 #3060  ; 針一狀態
OR<>(305) D320 #3060  ; 針二狀態
OR<>(305) D330 #3060  ; 針三狀態
ANDLD
LD W303.01  ; UV分數取樣中
LD<>(305) D313 #0  ; 針一分數高位
OR<>(305) D314 #0  ; 針一分數低位
AND=(300) D310 #3040  ; 針一狀態
LD<>(305) D323 #0  ; 針二分數高位
OR<>(305) D324 #0  ; 針二分數低位
AND=(300) D320 #3040  ; 針二狀態
ORLD
LD<>(305) D333 #0  ; 針三分數高位
OR<>(305) D334 #0  ; 針三分數低位
AND=(300) D330 #3040  ; 針三狀態
ORLD
ANDLD
ORLD
ANDLD
OUT W303.01  ; UV分數取樣中
LD TR0
%LD W303.01  ; UV分數取樣中
OR W303.02  ; UV分數取樣完成
ANDLD
OUT W303.02  ; UV分數取樣完成
@MOV(021) #0 D313  ; 針一分數高位
@MOV(021) #0 D314  ; 針一分數低位
@MOV(021) #0 D315  ; 針一指令傳送成功
@MOV(021) #0 D323  ; 針二分數高位
@MOV(021) #0 D324  ; 針二分數低位
@MOV(021) #0 D325  ; 針二指令傳送成功
@MOV(021) #0 D333  ; 針三分數高位
@MOV(021) #0 D334  ; 針三分數低位
@MOV(021) #0 D335  ; 針三指令傳送成功

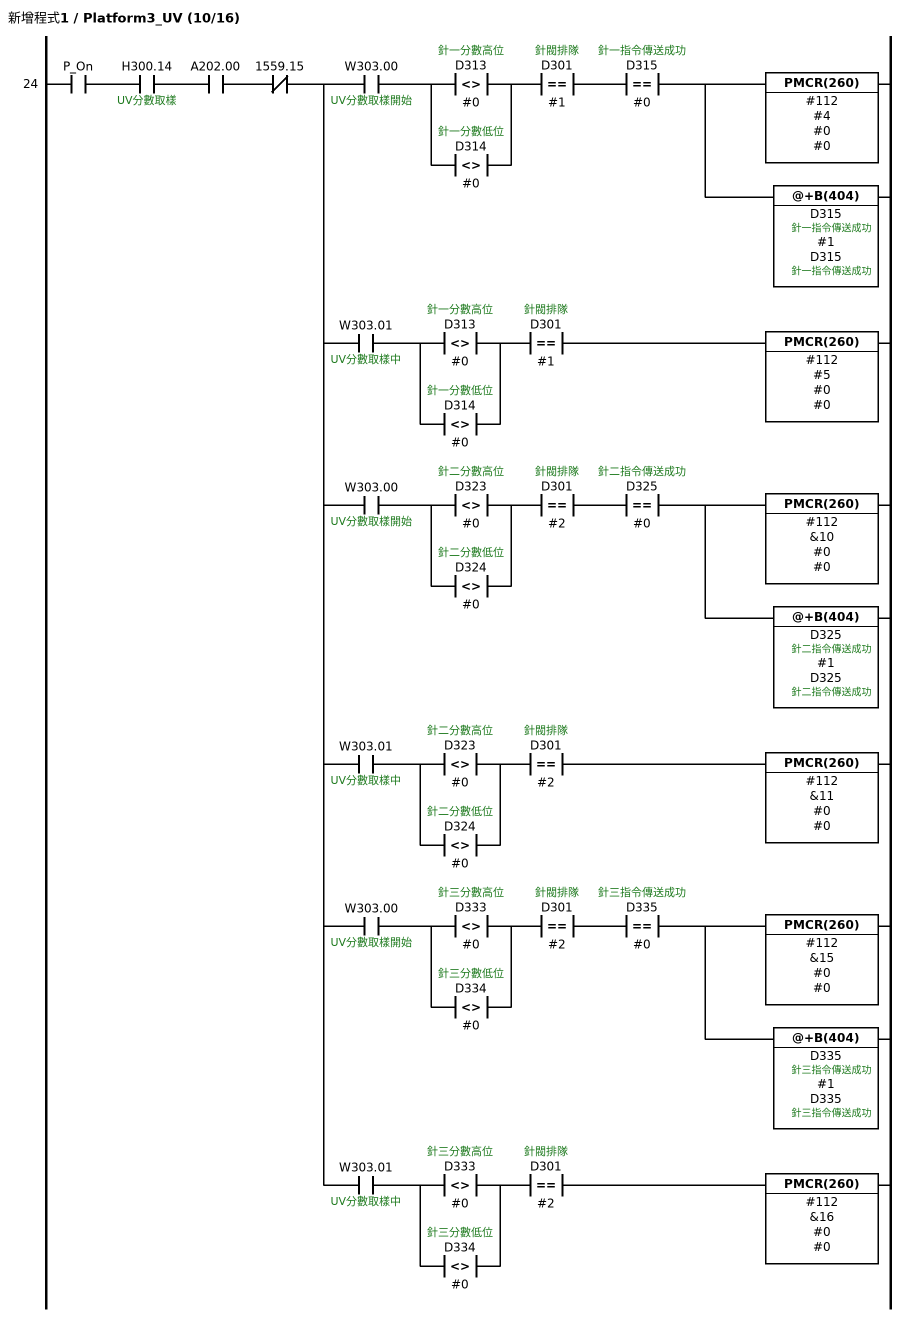
; rung 24
LD P_On
AND H300.14  ; UV分數取樣
AND A202.00
ANDNOT 1559.15
OUT TR0
AND W303.00  ; UV分數取樣開始
LD<>(305) D313 #0  ; 針一分數高位
OR<>(305) D314 #0  ; 針一分數低位
ANDLD
AND=(300) D301 #1  ; 針閥排隊
AND=(300) D315 #0  ; 針一指令傳送成功
PMCR(260) #112 #4 #0 #0
@+B(404) D315 #1 D315  ; 針一指令傳送成功
LD TR0
AND W303.01  ; UV分數取樣中
LD<>(305) D313 #0  ; 針一分數高位
OR<>(305) D314 #0  ; 針一分數低位
ANDLD
AND=(300) D301 #1  ; 針閥排隊
PMCR(260) #112 #5 #0 #0
LD TR0
AND W303.00  ; UV分數取樣開始
LD<>(305) D323 #0  ; 針二分數高位
OR<>(305) D324 #0  ; 針二分數低位
ANDLD
AND=(300) D301 #2  ; 針閥排隊
AND=(300) D325 #0  ; 針二指令傳送成功
PMCR(260) #112 &10 #0 #0
@+B(404) D325 #1 D325  ; 針二指令傳送成功
LD TR0
AND W303.01  ; UV分數取樣中
LD<>(305) D323 #0  ; 針二分數高位
OR<>(305) D324 #0  ; 針二分數低位
ANDLD
AND=(300) D301 #2  ; 針閥排隊
PMCR(260) #112 &11 #0 #0
LD TR0
AND W303.00  ; UV分數取樣開始
LD<>(305) D333 #0  ; 針三分數高位
OR<>(305) D334 #0  ; 針三分數低位
ANDLD
AND=(300) D301 #2  ; 針閥排隊
AND=(300) D335 #0  ; 針三指令傳送成功
PMCR(260) #112 &15 #0 #0
@+B(404) D335 #1 D335  ; 針三指令傳送成功
LD TR0
AND W303.01  ; UV分數取樣中
LD<>(305) D333 #0  ; 針三分數高位
OR<>(305) D334 #0  ; 針三分數低位
ANDLD
AND=(300) D301 #2  ; 針閥排隊
PMCR(260) #112 &16 #0 #0

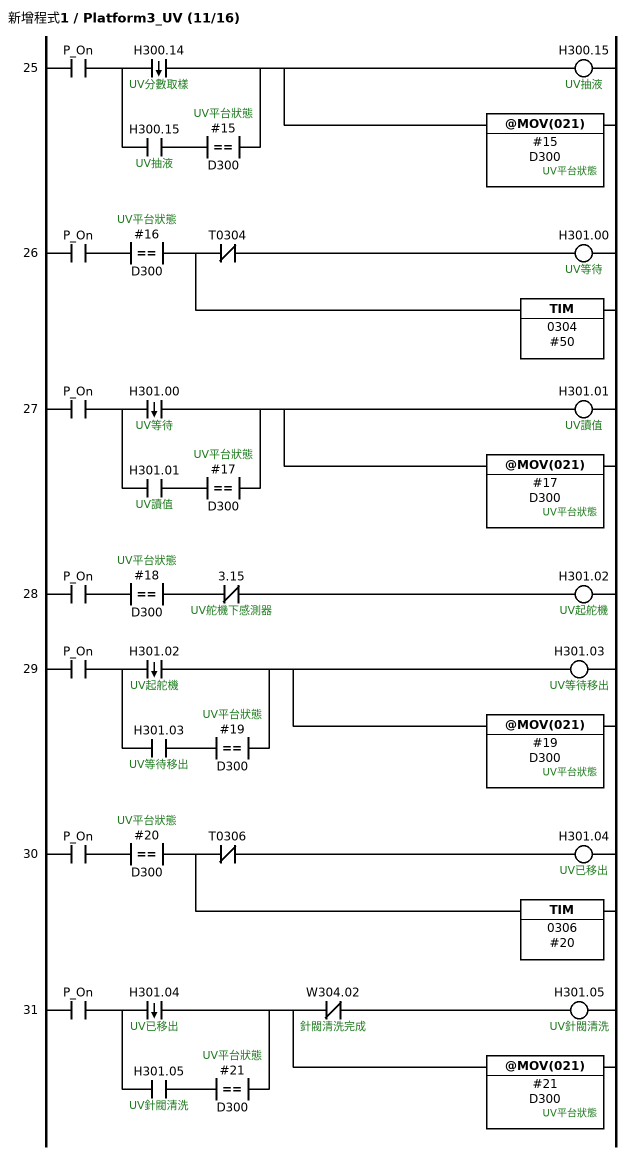
; rung 25
LD P_On
%LD H300.14  ; UV分數取樣
LD H300.15  ; UV抽液
AND=(300) #15 D300  ; UV平台狀態
ORLD
ANDLD
OUT H300.15  ; UV抽液
@MOV(021) #15 D300  ; UV平台狀態
; rung 26
LD P_On
AND=(300) #16 D300  ; UV平台狀態
OUT TR0
ANDNOT T0304
OUT H301.00  ; UV等待
LD TR0
TIM 0304 #50
; rung 27
LD P_On
%LD H301.00  ; UV等待
LD H301.01  ; UV讀值
AND=(300) #17 D300  ; UV平台狀態
ORLD
ANDLD
OUT H301.01  ; UV讀值
@MOV(021) #17 D300  ; UV平台狀態
; rung 28
LD P_On
AND=(300) #18 D300  ; UV平台狀態
ANDNOT 3.15  ; UV舵機下感測器
OUT H301.02  ; UV起舵機
; rung 29
LD P_On
%LD H301.02  ; UV起舵機
LD H301.03  ; UV等待移出
AND=(300) #19 D300  ; UV平台狀態
ORLD
ANDLD
OUT H301.03  ; UV等待移出
@MOV(021) #19 D300  ; UV平台狀態
; rung 30
LD P_On
AND=(300) #20 D300  ; UV平台狀態
OUT TR0
ANDNOT T0306
OUT H301.04  ; UV已移出
LD TR0
TIM 0306 #20
; rung 31
LD P_On
%LD H301.04  ; UV已移出
LD H301.05  ; UV針閥清洗
AND=(300) #21 D300  ; UV平台狀態
ORLD
ANDLD
OUT TR0
ANDNOT W304.02  ; 針閥清洗完成
OUT H301.05  ; UV針閥清洗
LD TR0
@MOV(021) #21 D300  ; UV平台狀態

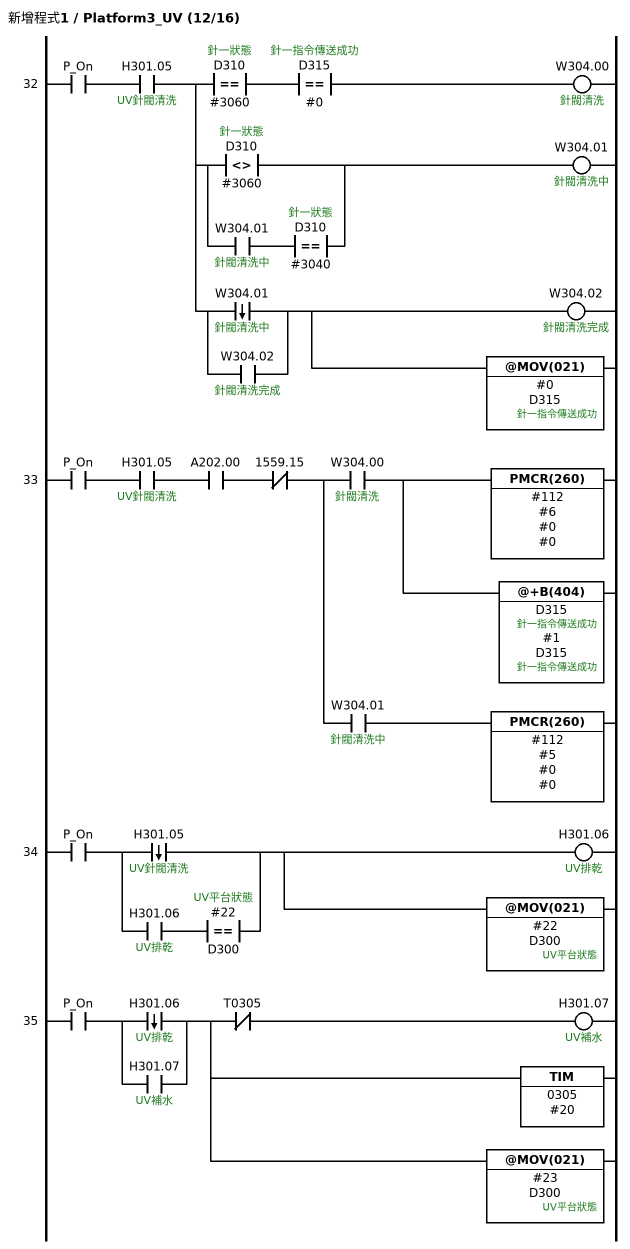
; rung 32
LD P_On
AND H301.05  ; UV針閥清洗
OUT TR0
AND=(300) D310 #3060  ; 針一狀態
AND=(300) D315 #0  ; 針一指令傳送成功
OUT W304.00  ; 針閥清洗
LD TR0
LD<>(305) D310 #3060  ; 針一狀態
LD W304.01  ; 針閥清洗中
AND=(300) D310 #3040  ; 針一狀態
ORLD
ANDLD
OUT W304.01  ; 針閥清洗中
LD TR0
%LD W304.01  ; 針閥清洗中
OR W304.02  ; 針閥清洗完成
ANDLD
OUT W304.02  ; 針閥清洗完成
@MOV(021) #0 D315  ; 針一指令傳送成功
; rung 33
LD P_On
AND H301.05  ; UV針閥清洗
AND A202.00
ANDNOT 1559.15
OUT TR0
AND W304.00  ; 針閥清洗
PMCR(260) #112 #6 #0 #0
@+B(404) D315 #1 D315  ; 針一指令傳送成功
LD TR0
AND W304.01  ; 針閥清洗中
PMCR(260) #112 #5 #0 #0
; rung 34
LD P_On
%LD H301.05  ; UV針閥清洗
LD H301.06  ; UV排乾
AND=(300) #22 D300  ; UV平台狀態
ORLD
ANDLD
OUT H301.06  ; UV排乾
@MOV(021) #22 D300  ; UV平台狀態
; rung 35
LD P_On
%LD H301.06  ; UV排乾
OR H301.07  ; UV補水
ANDLD
OUT TR0
ANDNOT T0305
OUT H301.07  ; UV補水
LD TR0
TIM 0305 #20
@MOV(021) #23 D300  ; UV平台狀態

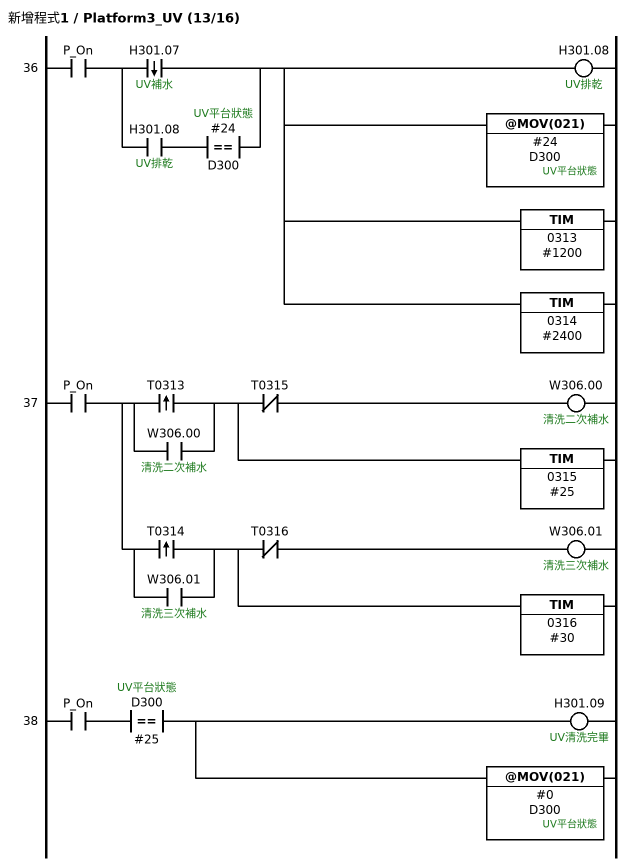
; rung 36
LD P_On
%LD H301.07  ; UV補水
LD H301.08  ; UV排乾
AND=(300) #24 D300  ; UV平台狀態
ORLD
ANDLD
OUT H301.08  ; UV排乾
@MOV(021) #24 D300  ; UV平台狀態
TIM 0313 #1200
TIM 0314 #2400
; rung 37
LD P_On
OUT TR0
@LD T0313
OR W306.00  ; 清洗二次補水
ANDLD
OUT TR1
ANDNOT T0315
OUT W306.00  ; 清洗二次補水
LD TR1
TIM 0315 #25
LD TR0
@LD T0314
OR W306.01  ; 清洗三次補水
ANDLD
OUT TR0
ANDNOT T0316
OUT W306.01  ; 清洗三次補水
LD TR0
TIM 0316 #30
; rung 38
LD P_On
AND=(300) D300 #25  ; UV平台狀態
OUT H301.09  ; UV清洗完畢
@MOV(021) #0 D300  ; UV平台狀態

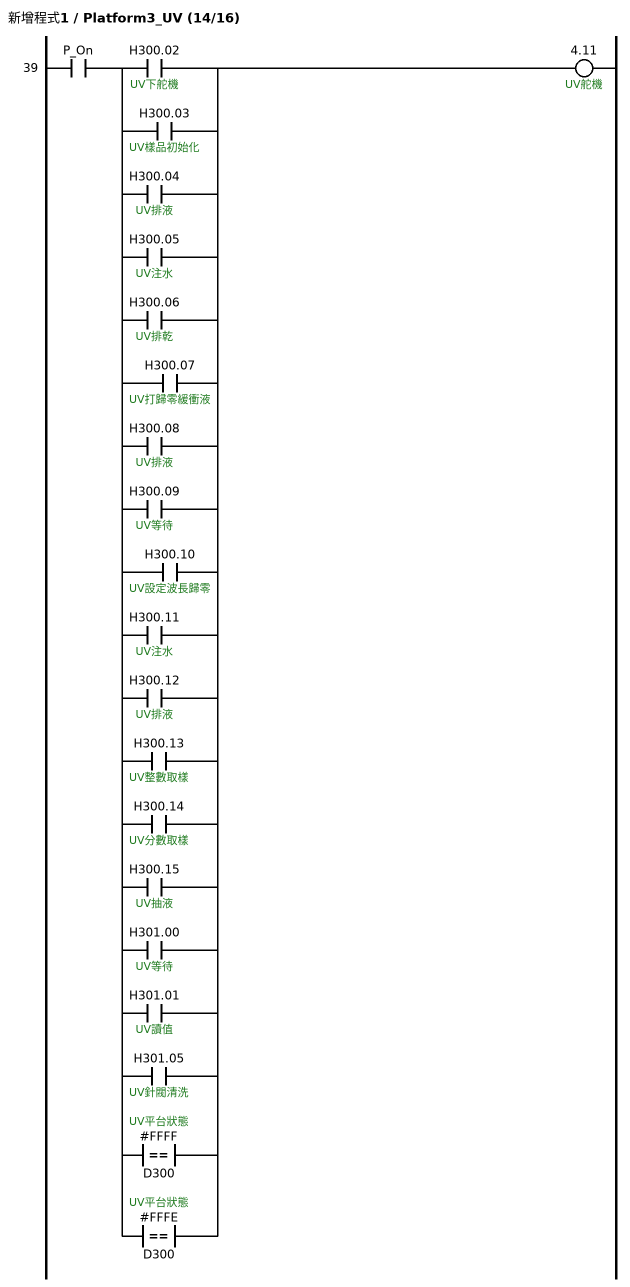
; rung 39
LD P_On
LD H300.02  ; UV下舵機
OR H300.03  ; UV樣品初始化
OR H300.04  ; UV排液
OR H300.05  ; UV注水
OR H300.06  ; UV排乾
OR H300.07  ; UV打歸零緩衝液
OR H300.08  ; UV排液
OR H300.09  ; UV等待
OR H300.10  ; UV設定波長歸零
OR H300.11  ; UV注水
OR H300.12  ; UV排液
OR H300.13  ; UV整數取樣
OR H300.14  ; UV分數取樣
OR H300.15  ; UV抽液
OR H301.00  ; UV等待
OR H301.01  ; UV讀值
OR H301.05  ; UV針閥清洗
OR=(300) #FFFF D300  ; UV平台狀態
OR=(300) #FFFE D300  ; UV平台狀態
ANDLD
OUT 4.11  ; UV舵機

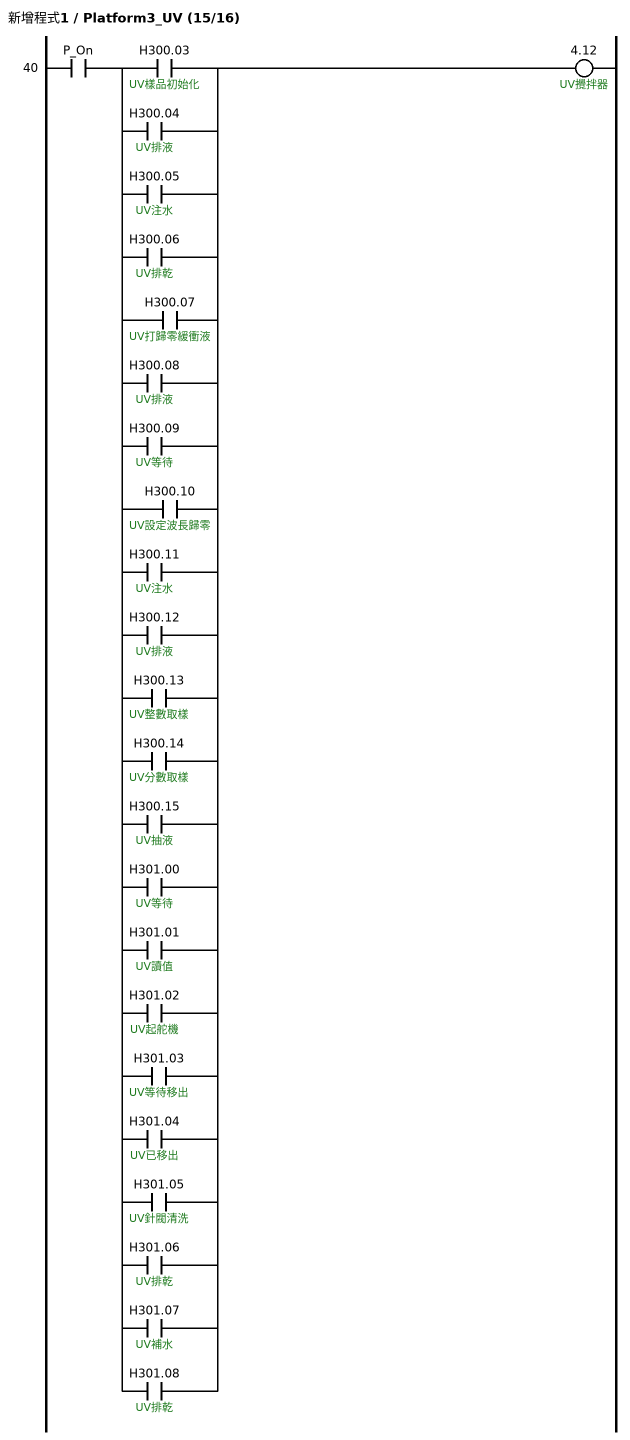
; rung 40
LD P_On
LD H300.03  ; UV樣品初始化
OR H300.04  ; UV排液
OR H300.05  ; UV注水
OR H300.06  ; UV排乾
OR H300.07  ; UV打歸零緩衝液
OR H300.08  ; UV排液
OR H300.09  ; UV等待
OR H300.10  ; UV設定波長歸零
OR H300.11  ; UV注水
OR H300.12  ; UV排液
OR H300.13  ; UV整數取樣
OR H300.14  ; UV分數取樣
OR H300.15  ; UV抽液
OR H301.00  ; UV等待
OR H301.01  ; UV讀值
OR H301.02  ; UV起舵機
OR H301.03  ; UV等待移出
OR H301.04  ; UV已移出
OR H301.05  ; UV針閥清洗
OR H301.06  ; UV排乾
OR H301.07  ; UV補水
OR H301.08  ; UV排乾
ANDLD
OUT 4.12  ; UV攪拌器

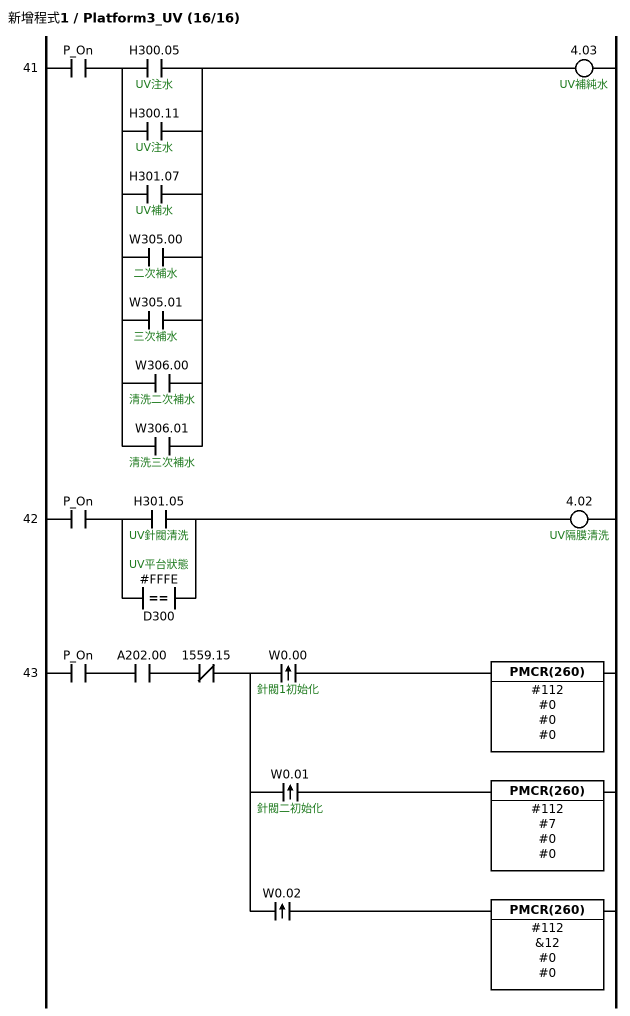
; rung 41
LD P_On
LD H300.05  ; UV注水
OR H300.11  ; UV注水
OR H301.07  ; UV補水
OR W305.00  ; 二次補水
OR W305.01  ; 三次補水
OR W306.00  ; 清洗二次補水
OR W306.01  ; 清洗三次補水
ANDLD
OUT 4.03  ; UV補純水
; rung 42
LD P_On
LD H301.05  ; UV針閥清洗
OR=(300) #FFFE D300  ; UV平台狀態
ANDLD
OUT 4.02  ; UV隔膜清洗
; rung 43
LD P_On
AND A202.00
ANDNOT 1559.15
OUT TR0
@AND W0.00  ; 針閥1初始化
PMCR(260) #112 #0 #0 #0
LD TR0
@AND W0.01  ; 針閥二初始化
PMCR(260) #112 #7 #0 #0
LD TR0
@AND W0.02
PMCR(260) #112 &12 #0 #0

### Section Seat

